(* IEC 61131-3 sources: ElnaAutomator/ExampleProject/build_USO_ecl (part 2) *)

  	END_CASE;
  END_IF;

  StrSw.Accident := inAccident.value AND inAccident.reliability;
  StrSw.Ns := inNs.value AND inNs.reliability;
  StrSw.Local := inLocal.value AND inLocal.reliability;
  StrSw.Distance := inDistance.value AND inDistance.reliability;
  StrSw.OpcCommandsDisabled := StrSw.inOpcCommandsDisabled;
  StrSw.offKNA := inoffKNA.value AND inoffKNA.reliability;

  (* ---- Формирование признака сдвига ---- *)

  getSdvig := FALSE;
  IF (StrSw.ISVALIDREF_cmdOn OR StrSw.ISVALIDREF_cmdOff) AND NOT StrSw.Local THEN
  	IF NOT (StrSw.CmdOn OR StrSw.CmdOff) THEN
                       IF (lastOnStatus <> StrSw.onStatus AND
  		(StrSw.onStatus <> _statusDualInput.STATUS_NOTDEFINED AND
                       StrSw.onStatus <> _statusDualInput.STATUS_ERROR)     AND
  		(lastOnStatus <> _statusDualInput.STATUS_NOTDEFINED   AND
                       lastOnStatus <> _statusDualInput.STATUS_ERROR))
                      THEN
  			getSdvig   := TRUE;
  		END_IF;
  	END_IF;
  END_IF;

  IF getSdvig THEN StrSw.sdvig:= TRUE; END_IF;

  sdvigReset(IN:=StrSw.sdvig, PT:=T#15S);

  IF sdvigReset.Q THEN StrSw.sdvig:=FALSE; END_IF;

  lastOnStatus := StrSw.onStatus;

  (* ---- Распаковка команды ---- *)
  _sunpackerCommand(command := StrSw.inCommand);
  	cmd := _sunpackerCommand.cmd;
  	source := _sunpackerCommand.source;

  (* ---- Обработка команды ---- *)
  IF cmd <> 0 AND lastCmd <> cmd and (((NOT StrSw.opcCommandsDisabled) AND source > 0) OR source = 0) then
  	CASE BYTE_TO_INT(cmd) OF
  	(*cmd_open*) 1 :
  			IF  StrSw.ISVALIDREF_cmdOn THEN StrSw.CmdOn := TRUE;
  				IF StrSw.ISVALIDREF_cmdOff THEN StrSw.CmdOff := FALSE; END_IF;
  			ELSIF  StrSw.ISVALIDREF_cmdOff THEN StrSw.CmdOff := FALSE;  END_IF;
  			errorCMDTimer(IN := false);
  			_commandErrorTimer := true;
  			StrSw.lastCmdIsOn := true;
  	(*cmd_close*) 2 :
  			IF StrSw.ISVALIDREF_cmdOff THEN StrSw.CmdOff := TRUE;
  				IF StrSw.ISVALIDREF_cmdOn THEN StrSw.CmdOn := FALSE; END_IF;
  			ELSIF StrSw.ISVALIDREF_cmdOn THEN StrSw.CmdOn := FALSE; END_IF;
  			errorCMDTimer(IN := false);
  			_commandErrorTimer := true;
  			StrSw.lastCmdIsOn := false;
  	(*cmd_reset*) 3 :    IF StrSw.ISVALIDREF_statOn OR StrSw.ISVALIDREF_statOff THEN
  			StrSw.CmdOn := FALSE;
  			StrSw.CmdOff := FALSE;
                                lastCmd := 0;
  			_commandErrorTimer := false;
  			StrSw.lastCmdIsOn := false;
                                 END_IF;
  	END_CASE;
  	source_for_Status := source;
  	cmd_for_Status := cmd;
  	command_error_for_Status := 0;
  END_IF;
  lastCmd := cmd;

  errorCMDTimer(In := _commandErrorTimer, PT :=T#10s);

  (* ---- алгоритм  для команды ВКЛючить ---- *)
  IF (StrSw.onStatus = _statusDualInput.STATUS_ON) and (StrSw.lastCmdIsOn) then
  	IF StrSw.ISVALIDREF_cmdOn AND StrSw.ISVALIDREF_cmdOff then  StrSw.cmdOn := false; END_IF;

  	 errorCMDTimer(In := false);
  	 _commandErrorTimer := false;
  	 cmd_for_Status := 0;
  	 source_for_Status := 0;
  END_IF;

  (* ---- off ---- *)
  IF (StrSw.onStatus = _statusDualInput.STATUS_OFF) and (NOT StrSw.lastCmdIsOn) then
  	IF StrSw.ISVALIDREF_cmdOn AND StrSw.ISVALIDREF_cmdOff then  StrSw.cmdOff := false; END_IF;

  	 errorCMDTimer(In := false);
  	 _commandErrorTimer := false;
  	 cmd_for_Status := 0;
  	 source_for_Status := 0;
  END_IF;

  (* ---- ошибка исполнения команды ---- *)
  if errorCMDTimer.Q and (cmd_for_Status <> 0) then
  	command_error_for_Status :=  cmd_for_Status;
  	_commandErrorTimer := false;
  	StrSw.CmdOn := false;
  	StrSw.CmdOff := false;
  	lastCmd := 0;
  end_if;

  (* ---- сброс ошибки команды ---- *)
  StrSw.CommandFault := command_error_for_Status <> 0;
  _errorReset(IN := command_error_for_Status <> 0, PT := T#5S);
  IF _errorReset.Q THEN
  	cmd_for_Status := 0;
  	source_for_Status := 0;
  	command_error_for_Status := 0;
  END_IF;

  outputsSets(in := (StrSw.ISVALIDREF_cmdOn and StrSw.cmdOn ) OR (StrSw.ISVALIDREF_cmdOff and StrSw.cmdOff), PT := T#2S);
  	IF NOT outputsSets.Q THEN
  		StrSw.BreakCmdOn := inBreakCmdOn._inversed AND inBreakCmdOn.reliability AND StrSw.ISVALIDREF_inBreakCmdOn;
  		StrSw.BreakCmdOff := inBreakCmdOff._inversed AND inBreakCmdOff.reliability AND StrSw.ISVALIDREF_inBreakCmdOff;
  	END_IF;

  cmdOn := StrSw.cmdOn;
  cmdOff:= StrSw.cmdOff;

  (* ---- формирование зашифрованного статуса для АРМа ---- *)
  StrSw.status := shl(BYTE_TO_DWORD(source_for_Status), 29)
  		OR shl(BYTE_TO_DWORD(cmd_for_Status), 26)
  		OR shl(BYTE_TO_DWORD(command_error_for_Status), 23)
  		OR shl(bool_to_DWORD(StrSw.sdvig), 22)
  		OR shl(bool_to_DWORD(StrSw.OpcCommandsDisabled), 21)
                      OR shl(BOOL_TO_DWORD(StrSw.offKNA), 17)
                      OR shl(bool_to_DWORD(StrSw.lastCmdIsOn), 14)
                      OR shl(BOOL_TO_DWORD(StrSw.BreakCmdOff), 13)
  		OR shl(BOOL_TO_DWORD(StrSw.BreakCmdOn), 12)
                      OR shl(BYTE_TO_DWORD(StrSw.basketStatus), 8)
  		OR shl(BOOL_TO_DWORD(StrSw.Distance), 6)
  		OR shl(BOOL_TO_DWORD(StrSw.Local), 5)
  		OR shl(BOOL_TO_DWORD(StrSw.Ns), 4)
                  	OR shl(BOOL_TO_DWORD(StrSw.Accident ),3)
  		OR BYTE_TO_DWORD(StrSw.onStatus);
END_FUNCTION_BLOCK

FUNCTION_BLOCK fb_singleOutput
  VAR_IN_OUT
    signal : BOOL;
    str_SO : struct_singleOutput;
  END_VAR
  VAR
    pulseTimer : TON;
    resetCmdTimer : TON;
    TON_Command : TON;
    source : BYTE;
    cmd : BYTE;
    lastCmd : BYTE;
    source_for_Status : BYTE;
    cmd_for_Status : BYTE;
    command_error_for_Status : BYTE;
    pulseTimerPriznak : BOOL;
    resetCmdTimerPriznak : BOOL;
    _sunpackerCommand : fb_sunpackerCommand;
  END_VAR

  str_SO.OpcCommandsDisabled := str_SO.inOpcCommandsDisabled;

  (* ---- Если управление с ВУ заблокировано, то передаем команду из алгоритма ---- *)
  IF str_SO.inOpcCommandsDisabled THEN
  	str_SO.inCommand := str_SO.inCommand_Alg;
  ELSE (* иначе передаем команду с АРМа*)
  	str_SO.inCommand := str_SO.inCommand_ARM;
  END_IF;

  (*Распаковка команды*)
  _sunpackerCommand(command := str_SO.inCommand);
  	cmd := _sunpackerCommand.cmd;
  	source := _sunpackerCommand.source;

  (*Обработка команды*)
  IF cmd <> 0 AND lastCmd <> cmd and (((NOT str_SO.OpcCommandsDisabled) AND source > 0) OR source = 0) then
  	CASE BYTE_TO_INT(cmd) OF
  	(*cmd_on*) 1 :
  			str_SO.Q := TRUE;
  			pulseTimer(IN := FALSE);
  			pulseTimerPriznak := FALSE;
  			resetCmdTimer(IN := FALSE);
  			resetCmdTimerPriznak := TRUE;
  	(*cmd_off*) 2 :
  			str_SO.Q := FALSE;
  			pulseTimer(IN := FALSE);
  			pulseTimerPriznak := FALSE;
  			resetCmdTimer(IN := FALSE);
  			resetCmdTimerPriznak := TRUE;
  	(*cmd_pulse*) 3 :
  			str_SO.Q := TRUE;
                                pulseTimer(IN := FALSE);
                                pulseTimerPriznak := TRUE;
  			resetCmdTimer(IN := FALSE);
                                resetCmdTimerPriznak := FALSE;
  	END_CASE;
  	source_for_Status := source;
  	cmd_for_Status := cmd;
  	command_error_for_Status := 0;
  END_IF;
  lastCmd := cmd;

  pulseTimer(IN := pulseTimerPriznak, PT := str_SO.wait_time);
  pulseTimer();
  IF pulseTimer.Q THEN
  	pulseTimer(IN := FALSE);
  	pulseTimerPriznak := FALSE;

  	str_SO.Q := FALSE;

  	source_for_Status := 0;
  	cmd_for_Status := 0;
  	command_error_for_Status := 0;
  END_IF;

  resetCmdTimer(IN := resetCmdTimerPriznak, PT := T#10S);
  resetCmdTimer();
  IF resetCmdTimer.Q THEN
  	resetCmdTimer(IN := FALSE);
  	resetCmdTimerPriznak := FALSE;

  	source_for_Status := 0;
  	cmd_for_Status := 0;
  	command_error_for_Status := 0;
  END_IF;

  signal:= str_SO.Q;

  (*TON_Command(IN:= (inCommand <> 0) AND (source = 0), PT:= T#2S);*)
      (*IF TON_Command.Q THEN*)
          (*inCommand := 0;*)
      (*END_IF;*)
  str_SO.status :=                           shl(BYTE_TO_DWORD(source_for_Status), 29)
  				OR shl(BYTE_TO_DWORD(cmd_for_Status), 26)
  				OR shl(BYTE_TO_DWORD(command_error_for_Status), 23)
  				OR shl(BOOL_TO_DWORD(str_SO.OpcCommandsDisabled), 21)
  				OR BOOL_TO_DWORD(str_SO.Q);
END_FUNCTION_BLOCK

FUNCTION_BLOCK fb_singleSignal
  VAR_INPUT
    signal : TYPE_ReliableBit;
  END_VAR
  VAR_IN_OUT
    str_SS : struct_singleSignal;
  END_VAR
  VAR
    TimerOn : TON;
    TimerOff : TOF;
  END_VAR

  str_SS.reliability:=signal.reliability;

  IF NOT str_SS.inverse THEN
  TimerOn(IN:=(signal.value AND str_SS.reliability AND NOT str_SS.Disabled_Sig), PT:=str_SS.DelayOn);
  ELSE
  TimerOn(IN:=(signal._inversed AND str_SS.reliability AND NOT str_SS.Disabled_Sig), PT:=str_SS.DelayOn);
  END_IF;

  TimerOff(IN:=TimerOn.Q, PT:=str_SS.DelayOff);

  str_SS.Q:=TimerOff.Q;

  str_SS.status:= SHL(BOOL_TO_DWORD(NOT str_SS.reliability), 15)
  	OR BOOL_TO_DWORD(str_SS.Q);
END_FUNCTION_BLOCK

FUNCTION_BLOCK Proc_Im
  VAR
    fb_Kran1 : fb_Kran;
    fb_Kran4 : fb_Kran;
    fb_Kran2 : fb_Kran;
    fb_Kran3 : fb_Kran;
    fb_Nu : fb_OilPump;
    fb_Nu2 : fb_OilPump;
    fb_Mv : fb_SectionSwitch;
    fb_SectionSwitch1 : fb_SectionSwitch;
    fb_Avom1 : fb_Switch;
    fb_Avom2 : fb_Switch;
    fb_Avom3 : fb_Switch;
    fb_Avom4 : fb_Switch;
    fb_So0 : fb_singleOutput;
    fb_So1 : fb_singleOutput;
    fb_So2 : fb_singleOutput;
    fb_So3 : fb_singleOutput;
    fb_So4 : fb_singleOutput;
    fb_So5 : fb_singleOutput;
    fb_So6 : fb_singleOutput;
    fb_So7 : fb_singleOutput;
    fb_SI0 : fb_singleSignal;
    fb_SI1 : fb_singleSignal;
    fb_SI2 : fb_singleSignal;
    fb_SI3 : fb_singleSignal;
    fb_SI4 : fb_singleSignal;
    fb_SI5 : fb_singleSignal;
    fb_SI6 : fb_singleSignal;
  END_VAR
  VAR_EXTERNAL
    di : DiConfig;
    od : DoConfig;
    Im : ImConfig;
  END_VAR

  fb_Kran1(statOn := di.Di.bits[1]._inversed,
  statOn_reliability := di.Di.bits[1].reliability,
  statOff := di.Di.bits[2]._inversed,
  statOff_reliability := di.Di.bits[2].reliability,
  cmdOn := od.Do1.bits[1],
  cmdOff := od.Do2.bits[0],
  inDp := di.Di1.bits[1],
  inSo := di.Di.bits[3],
  inSz := di.Di.bits[2],
  strKr := Im.Kran1);

  fb_Kran4(statOn := di.Di1.bits[2]._inversed,
  statOn_reliability := di.Di1.bits[2].reliability,
  statOff := di.Di2.bits[2]._inversed,
  statOff_reliability := di.Di2.bits[2].reliability,
  cmdOn := od.Do3.bits[2],
  cmdOff := od.Do1.bits[2],
  inDp := di.Di.bits[2],
  inSo := di.Di2.bits[3],
  inSz := di.Di1.bits[1],
  strKr := Im.Kran4);

  fb_Kran2(statOn := di.Di2.bits[3].value,
  statOn_reliability := di.Di2.bits[3].reliability,
  statOff := di.Di3.bits[1].value,
  statOff_reliability := di.Di3.bits[1].reliability,
  cmdOn := od.Do3.bits[3],
  cmdOff := od.Do2.bits[3],
  inDp := di.Di4.bits[3],
  inSo := di.Di1.bits[1],
  inSz := di.Di1.bits[2],
  strKr := Im.Kran2);

  fb_Kran3(statOn := di.Di3.bits[4]._inversed,
  statOn_reliability := di.Di3.bits[4].reliability,
  statOff := di.Di4.bits[3]._inversed,
  statOff_reliability := di.Di4.bits[3].reliability,
  cmdOn := od.Do2.bits[4],
  cmdOff := od.Do3.bits[4],
  inDp := di.Di4.bits[4],
  inSo := di.Di1.bits[2],
  inSz := di.Di4.bits[3],
  strKr := Im.Kran3);

  fb_Nu(statOn := di.Di.bits[1]._inversed,
  statOn_reliability := di.Di.bits[1].reliability,
  statOff := di.Di.bits[2]._inversed,
  statOff_reliability := di.Di.bits[2].reliability,
  cmdOn := od.Do2.bits[1],
  cmdOff := od.Do1.bits[0],
  inBreakCmdOn := di.Di.bits[3],
  inBreakCmdOff := di.Di1.bits[4],
  StrSw := Im.Nu);

  fb_Nu2(statOn := di.Di2.bits[2].value,
  statOn_reliability := di.Di2.bits[2].reliability,
  statOff := di.Di3.bits[3].value,
  statOff_reliability := di.Di3.bits[3].reliability,
  cmdOn := od.Do4.bits[3],
  cmdOff := od.Do1.bits[4],
  inBreakCmdOn := di.Di.bits[4],
  inBreakCmdOff := di.Di1.bits[3],
  StrSw := Im.Nu2);

  fb_Avom1(statOn := di.Di.bits[1].value,
  statOn_reliability := di.Di.bits[1].reliability,
  statOff := di.Di1.bits[2].value,
  statOff_reliability := di.Di1.bits[2].reliability,
  cmdOn := od.Do1.bits[1],
  cmdOff := od.Do1.bits[0],
  inBreakCmdOn := di.Di1.bits[2],
  inBreakCmdOff := di.Di.bits[2],
  StrSw := Im.Avom1);

  fb_Avom2(statOn := di.Di3.bits[2]._inversed,
  statOn_reliability := di.Di3.bits[2].reliability,
  statOff := di.Di.bits[2]._inversed,
  statOff_reliability := di.Di.bits[2].reliability,
  cmdOn := od.Do4.bits[3],
  cmdOff := od.Do2.bits[1],
  inBreakCmdOn := di.Di1.bits[3],
  inBreakCmdOff := di.Di1.bits[3],
  StrSw := Im.Avom2);

  fb_Avom3(statOn := di.Di1.bits[3]._inversed,
  statOn_reliability := di.Di1.bits[3].reliability,
  statOff := di.Di2.bits[3]._inversed,
  statOff_reliability := di.Di2.bits[3].reliability,
  cmdOn := od.Do1.bits[5],
  cmdOff := od.Do3.bits[3],
  inBreakCmdOn := di.Di3.bits[4],
  inBreakCmdOff := di.Di2.bits[4],
  StrSw := Im.Avom3);

  fb_Avom4(statOn := di.Di.bits[4]._inversed,
  statOn_reliability := di.Di.bits[4].reliability,
  statOff := di.Di.bits[4]._inversed,
  statOff_reliability := di.Di.bits[4].reliability,
  cmdOn := od.Do2.bits[4],
  cmdOff := od.Do3.bits[4],
  inBreakCmdOn := di.Di3.bits[5],
  inBreakCmdOff := di.Di4.bits[5],
  StrSw := Im.Avom4);

  fb_Mv(statOn := di.Di.bits[1]._inversed,
  statOn_reliability := di.Di.bits[1].reliability,
  statOff := di.Di.bits[2]._inversed,
  statOff_reliability := di.Di.bits[2].reliability,
  cmdOn := od.Do2.bits[1],
  cmdOff := od.Do2.bits[0],
  inBreakCmdOn := di.Di3.bits[4],
  inBreakCmdOff := di.Di4.bits[3],
  basketRolledin := di.Di.bits[2],
  basketRolledout := di.Di.bits[3],
  basketTest := di.Di1.bits[3],
  StrSw := Im.Mv);

  fb_SectionSwitch1(StrSw := Im.SectionSwitch1);

  fb_SI0(signal := di.Di1.bits[1], str_SS := Im.SingleSignals.SI0);

  fb_SI1(signal := di.Di1.bits[2], str_SS := Im.SingleSignals.SI1);

  fb_SI2(signal := di.Di.bits[3], str_SS := Im.SingleSignals.SI2);

  fb_SI3(signal := di.Di1.bits[4], str_SS := Im.SingleSignals.SI3);

  fb_SI4(signal := di.Di3.bits[5], str_SS := Im.SingleSignals.SI4);

  fb_SI5(signal := di.Di3.bits[6], str_SS := Im.SingleSignals.SI5);

  fb_SI6(signal := di.Di4.bits[7], str_SS := Im.SingleSignals.SI6);

  fb_So0(signal := od.Do1.bits[1], str_SO := Im.SingleOutputs.So0);

  fb_So1(signal := od.Do2.bits[2], str_SO := Im.SingleOutputs.So1);

  fb_So2(signal := od.Do3.bits[3], str_SO := Im.SingleOutputs.So2);

  fb_So3(signal := od.Do1.bits[4], str_SO := Im.SingleOutputs.So3);

  fb_So4(signal := od.Do2.bits[5], str_SO := Im.SingleOutputs.So4);

  fb_So5(signal := od.Do1.bits[6], str_SO := Im.SingleOutputs.So5);

  fb_So6(signal := od.Do1.bits[7], str_SO := Im.SingleOutputs.So6);

  fb_So7(signal := od.Do2.bits[8], str_SO := Im.SingleOutputs.So7);
END_FUNCTION_BLOCK

FUNCTION_BLOCK Proc_Do_Init
  VAR_INPUT
    init : BOOL;
  END_VAR
  VAR
    stDO_Ini : fb_DO_Init;
    inits : UINT;
  END_VAR
  VAR_INPUT
    initiales : UINT;
  END_VAR
  VAR_EXTERNAL
    od : DoConfig;
  END_VAR

  inits := 0;

  stDO_Ini(data_Ini := TRUE, imit := FALSE, strDO := od.Do1);
  inits := inits + BOOL_TO_UINT(stDO_Ini.Init);

  stDO_Ini(data_Ini := TRUE, imit := FALSE, strDO := od.Do2);
  inits := inits + BOOL_TO_UINT(stDO_Ini.Init);

  stDO_Ini(data_Ini := TRUE, imit := FALSE, strDO := od.Do3);
  inits := inits + BOOL_TO_UINT(stDO_Ini.Init);

  stDO_Ini(data_Ini := TRUE, imit := FALSE, strDO := od.Do4);
  inits := inits + BOOL_TO_UINT(stDO_Ini.Init);

  stDO_Ini(data_Ini := TRUE, imit := FALSE, strDO := od.Do5);
  inits := inits + BOOL_TO_UINT(stDO_Ini.Init);

  initiales := 0;
  IF init THEN initiales := inits; END_IF;
END_FUNCTION_BLOCK

FUNCTION_BLOCK Opc_Im_set
  VAR_EXTERNAL
    Im : ImConfig;
    Im_Kran1_status : UDINT;
    Im_Kran4_status : UDINT;
    Im_Kran2_status : UDINT;
    Im_Kran3_status : UDINT;
    Im_Nu_status : UDINT;
    Im_Nu2_status : UDINT;
    Im_Avom1_status : UDINT;
    Im_Avom2_status : UDINT;
    Im_Avom3_status : UDINT;
    Im_Avom4_status : UDINT;
    Im_Mv_status : UDINT;
    Im_SectionSwitch1_status : UDINT;
    Im_SingleSignals_SI0_status : UDINT;
    Im_SingleSignals_SI1_status : UDINT;
    Im_SingleSignals_SI2_status : UDINT;
    Im_SingleSignals_SI3_status : UDINT;
    Im_SingleSignals_SI4_status : UDINT;
    Im_SingleSignals_SI5_status : UDINT;
    Im_SingleSignals_SI6_status : UDINT;
  END_VAR

  Im_Kran1_status := DWORD_TO_UDINT(Im.Kran1.status);

  Im_Kran4_status := DWORD_TO_UDINT(Im.Kran4.status);

  Im_Kran2_status := DWORD_TO_UDINT(Im.Kran2.status);

  Im_Kran3_status := DWORD_TO_UDINT(Im.Kran3.status);

  Im_Nu_status := DWORD_TO_UDINT(Im.Nu.status);

  Im_Nu2_status := DWORD_TO_UDINT(Im.Nu2.status);

  Im_Avom1_status := DWORD_TO_UDINT(Im.Avom1.status);

  Im_Avom2_status := DWORD_TO_UDINT(Im.Avom2.status);

  Im_Avom3_status := DWORD_TO_UDINT(Im.Avom3.status);

  Im_Avom4_status := DWORD_TO_UDINT(Im.Avom4.status);

  Im_Mv_status := DWORD_TO_UDINT(Im.Mv.status);

  Im_SectionSwitch1_status := DWORD_TO_UDINT(Im.SectionSwitch1.status);

  Im_SingleSignals_SI0_status := DWORD_TO_UDINT(Im.SingleSignals.SI0.status);

  Im_SingleSignals_SI1_status := DWORD_TO_UDINT(Im.SingleSignals.SI1.status);

  Im_SingleSignals_SI2_status := DWORD_TO_UDINT(Im.SingleSignals.SI2.status);

  Im_SingleSignals_SI3_status := DWORD_TO_UDINT(Im.SingleSignals.SI3.status);

  Im_SingleSignals_SI4_status := DWORD_TO_UDINT(Im.SingleSignals.SI4.status);

  Im_SingleSignals_SI5_status := DWORD_TO_UDINT(Im.SingleSignals.SI5.status);

  Im_SingleSignals_SI6_status := DWORD_TO_UDINT(Im.SingleSignals.SI6.status);
END_FUNCTION_BLOCK

FUNCTION_BLOCK Opc_Im_get
  VAR_EXTERNAL
    Im : ImConfig;
    Im_Kran1_inCommand_ARM : UINT;
    Im_Kran4_inCommand_ARM : UINT;
    Im_Kran2_inCommand_ARM : UINT;
    Im_Kran3_inCommand_ARM : UINT;
    Im_Nu_inCommand_ARM : UINT;
    Im_Nu2_inCommand_ARM : UINT;
    Im_Avom1_inCommand_ARM : UINT;
    Im_Avom2_inCommand_ARM : UINT;
    Im_Avom3_inCommand_ARM : UINT;
    Im_Avom4_inCommand_ARM : UINT;
    Im_Mv_inCommand_ARM : UINT;
    Im_SectionSwitch1_inCommand_ARM : UINT;
  END_VAR

  Im.Kran1.inCommand_ARM := UINT_TO_WORD(Im_Kran1_inCommand_ARM);

  Im.Kran4.inCommand_ARM := UINT_TO_WORD(Im_Kran4_inCommand_ARM);

  Im.Kran2.inCommand_ARM := UINT_TO_WORD(Im_Kran2_inCommand_ARM);

  Im.Kran3.inCommand_ARM := UINT_TO_WORD(Im_Kran3_inCommand_ARM);

  Im.Nu.inCommand_ARM := UINT_TO_WORD(Im_Nu_inCommand_ARM);

  Im.Nu2.inCommand_ARM := UINT_TO_WORD(Im_Nu2_inCommand_ARM);

  Im.Avom1.inCommand_ARM := UINT_TO_WORD(Im_Avom1_inCommand_ARM);

  Im.Avom2.inCommand_ARM := UINT_TO_WORD(Im_Avom2_inCommand_ARM);

  Im.Avom3.inCommand_ARM := UINT_TO_WORD(Im_Avom3_inCommand_ARM);

  Im.Avom4.inCommand_ARM := UINT_TO_WORD(Im_Avom4_inCommand_ARM);

  Im.Mv.inCommand_ARM := UINT_TO_WORD(Im_Mv_inCommand_ARM);

  Im.SectionSwitch1.inCommand_ARM := UINT_TO_WORD(Im_SectionSwitch1_inCommand_ARM);
END_FUNCTION_BLOCK

FUNCTION_BLOCK Opc_Ai_set
  VAR_EXTERNAL
    Ai : AiConfig;
    AI_A1_HW : LREAL;
    AI_A1_HA : LREAL;
    AI_A1_LA : LREAL;
    AI_A1_LW : LREAL;
    AI_A1_HL : LREAL;
    AI_A1_LL : LREAL;
    AI_A1_value : LREAL;
    AI_A1_status : UDINT;
    AI_A2_HW : LREAL;
    AI_A2_HA : LREAL;
    AI_A2_LA : LREAL;
    AI_A2_LW : LREAL;
    AI_A2_HL : LREAL;
    AI_A2_LL : LREAL;
    AI_A2_value : LREAL;
    AI_A2_status : UDINT;
  END_VAR

  AI_A1_HW := Ai.A1.HW;
  AI_A1_HA := Ai.A1.HA;
  AI_A1_LA := Ai.A1.LA;
  AI_A1_LW := Ai.A1.LW;
  AI_A1_LL := Ai.A1.LL;
  AI_A1_HL := Ai.A1.HL;
  AI_A1_value := Ai.A1.value;
  AI_A1_status := DWORD_TO_UDINT(Ai.A1.status);

  AI_A2_HW := Ai.A2.HW;
  AI_A2_HA := Ai.A2.HA;
  AI_A2_LA := Ai.A2.LA;
  AI_A2_LW := Ai.A2.LW;
  AI_A2_LL := Ai.A2.LL;
  AI_A2_HL := Ai.A2.HL;
  AI_A2_value := Ai.A2.value;
  AI_A2_status := DWORD_TO_UDINT(Ai.A2.status);
END_FUNCTION_BLOCK

FUNCTION_BLOCK Proc_Do
  VAR
    fb_Do1 : fb_DOSourceMlp;
    fb_Do2 : fb_DOSourceMlp;
    fb_Do3 : fb_DOSourceMlp;
    fb_Do4 : fb_DOSourceMlp;
    fb_Do5 : fb_DOSourceMlp;
  END_VAR
  VAR_EXTERNAL
    od : DoConfig;
    arDOUT_0 : TWordData;
    arDOUT_1 : TWordData;
    arDOUT_2 : TWordData;
    arDOUT_3 : TWordData;
    arDOUT_4 : TWordData;
    DO_0_wValue : UINT;
    DO_1_wValue : UINT;
    DO_2_wValue : UINT;
    DO_3_wValue : UINT;
    DO_4_wValue : UINT;
    arERR_1 : TItemDIN;
    arERR_2 : TItemDIN;
    arERR_3 : TItemDIN;
    arERR_4 : TItemDIN;
    arERR_5 : TItemDIN;
  END_VAR

  fb_Do1(arDout := arDOUT_0, strDO := od.Do1, err_mod := arERR_1);
  DO_0_wValue := arDOUT_0.wValue;

  fb_Do2(arDout := arDOUT_1, strDO := od.Do2, err_mod := arERR_2);
  DO_1_wValue := arDOUT_1.wValue;

  fb_Do3(arDout := arDOUT_2, strDO := od.Do3, err_mod := arERR_3);
  DO_2_wValue := arDOUT_2.wValue;

  fb_Do4(arDout := arDOUT_3, strDO := od.Do4, err_mod := arERR_4);
  DO_3_wValue := arDOUT_3.wValue;

  fb_Do5(arDout := arDOUT_4, strDO := od.Do5, err_mod := arERR_5);
  DO_4_wValue := arDOUT_4.wValue;

  (*gpio_out not initialized*)
END_FUNCTION_BLOCK

FUNCTION_BLOCK Proc_Di_Init
  VAR_INPUT
    init : BOOL;
  END_VAR
  VAR
    stDI_Ini : fb_DI_Init;
    inits : UINT;
  END_VAR
  VAR_INPUT
    initiales : UINT;
  END_VAR
  VAR_EXTERNAL
    di : DiConfig;
  END_VAR

  inits := 0;

  stDI_Ini(data_Ini := TRUE, imit := FALSE, strDI := di.Di);
  inits := inits + BOOL_TO_UINT(stDI_Ini.Init);

  stDI_Ini(data_Ini := TRUE, imit := FALSE, strDI := di.Di1);
  inits := inits + BOOL_TO_UINT(stDI_Ini.Init);

  stDI_Ini(data_Ini := TRUE, imit := FALSE, strDI := di.Di2);
  inits := inits + BOOL_TO_UINT(stDI_Ini.Init);

  stDI_Ini(data_Ini := TRUE, imit := FALSE, strDI := di.Di3);
  inits := inits + BOOL_TO_UINT(stDI_Ini.Init);

  stDI_Ini(data_Ini := TRUE, imit := FALSE, strDI := di.Di4);
  inits := inits + BOOL_TO_UINT(stDI_Ini.Init);

  initiales := 0;
  IF init THEN initiales := inits; END_IF;
END_FUNCTION_BLOCK

FUNCTION_BLOCK Opc_Protections_set
  VAR_EXTERNAL
    Protections : ProtectionsConfig;
    Protections_Ap1_status : UDINT;
    Protections_AiP1_status : UDINT;
    Protections_AiP2_status : UDINT;
    Protections_AiP3_status : UDINT;
    Protections_DiP1_status : UDINT;
    Protections_DiP2_status : UDINT;
    Protections_DiP3_status : UDINT;
    Protections_DiP4_status : UDINT;
    Protections_DiP5_status : UDINT;
  END_VAR

  Protections_Ap1_status := DWORD_TO_UDINT(Protections.Ap1.status);

  Protections_AiP1_status := DWORD_TO_UDINT(Protections.AiP1.status);

  Protections_AiP2_status := DWORD_TO_UDINT(Protections.AiP2.status);

  Protections_AiP3_status := DWORD_TO_UDINT(Protections.AiP3.status);

  Protections_DiP1_status := DWORD_TO_UDINT(Protections.DiP1.status);

  Protections_DiP2_status := DWORD_TO_UDINT(Protections.DiP2.status);

  Protections_DiP3_status := DWORD_TO_UDINT(Protections.DiP3.status);

  Protections_DiP4_status := DWORD_TO_UDINT(Protections.DiP4.status);

  Protections_DiP5_status := DWORD_TO_UDINT(Protections.DiP5.status);
END_FUNCTION_BLOCK

FUNCTION_BLOCK Opc_Protections_get
  VAR_EXTERNAL
    Protections : ProtectionsConfig;
    Protections_Ap1_inCommand_ARM : UINT;
    Protections_AiP1_inCommand_ARM : UINT;
    Protections_AiP2_inCommand_ARM : UINT;
    Protections_AiP3_inCommand_ARM : UINT;
    Protections_DiP1_inCommand_ARM : UINT;
    Protections_DiP2_inCommand_ARM : UINT;
    Protections_DiP3_inCommand_ARM : UINT;
    Protections_DiP4_inCommand_ARM : UINT;
    Protections_DiP5_inCommand_ARM : UINT;
  END_VAR

  Protections.Ap1.inCommand_ARM := UINT_TO_WORD(Protections_Ap1_inCommand_ARM);

  Protections.AiP1.inCommand_ARM := UINT_TO_WORD(Protections_AiP1_inCommand_ARM);

  Protections.AiP2.inCommand_ARM := UINT_TO_WORD(Protections_AiP2_inCommand_ARM);

  Protections.AiP3.inCommand_ARM := UINT_TO_WORD(Protections_AiP3_inCommand_ARM);

  Protections.DiP1.inCommand_ARM := UINT_TO_WORD(Protections_DiP1_inCommand_ARM);

  Protections.DiP2.inCommand_ARM := UINT_TO_WORD(Protections_DiP2_inCommand_ARM);

  Protections.DiP3.inCommand_ARM := UINT_TO_WORD(Protections_DiP3_inCommand_ARM);

  Protections.DiP4.inCommand_ARM := UINT_TO_WORD(Protections_DiP4_inCommand_ARM);

  Protections.DiP5.inCommand_ARM := UINT_TO_WORD(Protections_DiP5_inCommand_ARM);
END_FUNCTION_BLOCK

FUNCTION_BLOCK fb_DiSourceMlp
  VAR_INPUT
    arDIN : TItemDIN;
    err_mod : TItemDIN;
  END_VAR
  VAR_IN_OUT
    strDI : struct_DI;
  END_VAR
  VAR_OUTPUT
    Bounce : BOOL;
  END_VAR
  VAR
    _value : WORD;
    _reliability : BOOL;
    bitNumber : INT;
    bitNum : INT;
  END_VAR

  strDI.blConnect := (*((UINT_TO_WORD(arDIN.wFlags) = 1472) and*) (UINT_TO_WORD(err_mod.wValue) = 20) and (UINT_TO_WORD(err_mod.wFlags) = 192);
  Bounce := (UINT_TO_WORD(arDIN.wFlags) AND 16#0020) <> 0;

  If NOT strDI.imit THEN
  _value:=UINT_TO_WORD(arDIN.wValue);

      IF strDI.blConnect THEN
            strDI.reliability:=0;
            strDI.value:=0;
  	FOR bitNumber:=0 TO 7 BY 1 DO

  		_reliability:=WORD_TO_BOOL(SHR(_value, bitNumber*2) AND 16#2);
  		strDI.reliability:=strDI.reliability OR SHL(BOOL_TO_WORD(_reliability),bitNumber);
  		IF _reliability THEN
  			strDI.value:=strDI.value OR SHL((SHR(_value, bitNumber*2) AND 16#1),bitNumber);
  		END_IF;
  	END_FOR;
      ELSE
  	strDI.reliability := 0;
      END_IF;

      FOR bitNum:=0 TO 15 BY 1 DO
  	          strDI.bits[bitNum].reliability :=WORD_TO_BOOL(SHR(strDI.reliability, bitNum) AND 16#1);
  	IF strDI.bits[bitNum].reliability THEN
  		strDI.bits[bitNum].value :=WORD_TO_BOOL(SHR(strDI.value, bitNum) AND 16#1);
                      strDI.bits[bitNum]._inversed :=NOT strDI.bits[bitNum].value;
  	END_IF;
      END_FOR;

  END_IF;
END_FUNCTION_BLOCK

FUNCTION_BLOCK Proc_Protections_Init
  VAR_INPUT
    init : BOOL;
  END_VAR
  VAR
    stDIp_Ini : fb_DiProtection_Init;
    stAIp_Ini : fb_AiProtection_Init;
    inits : UINT;
  END_VAR
  VAR_INPUT
    initiales : UINT;
  END_VAR
  VAR_EXTERNAL
    Protections : ProtectionsConfig;
  END_VAR
  VAR
    _ProtectionTags : TYPE_ProtectionTags;
    _StatusAi : TYPE_StatusAi;
  END_VAR

  inits := 0;

  stAIp_Ini(data_Ini := TRUE, delay := T#1S, inTag := _ProtectionTags.AOS, inRunOnStart := TRUE,
  controlLimit := _StatusAi.LA, str_AIp := Protections.Ap1);
  inits := inits + BOOL_TO_UINT(stAIp_Ini.Init);

  stAIp_Ini(data_Ini := TRUE, delay := T#2S, inTag := _ProtectionTags.AOS, inRunOnStart := FALSE,
  controlLimit := _StatusAi.HA, str_AIp := Protections.AiP1);
  inits := inits + BOOL_TO_UINT(stAIp_Ini.Init);

  stAIp_Ini(data_Ini := TRUE, delay := T#3S, inTag := _ProtectionTags.AOS, inRunOnStart := TRUE,
  controlLimit := _StatusAi.LA, str_AIp := Protections.AiP2);
  inits := inits + BOOL_TO_UINT(stAIp_Ini.Init);

  stAIp_Ini(data_Ini := TRUE, delay := T#4S, inTag := _ProtectionTags.AOS, inRunOnStart := FALSE,
  controlLimit := _StatusAi.HA, str_AIp := Protections.AiP3);
  inits := inits + BOOL_TO_UINT(stAIp_Ini.Init);

  stDIp_Ini(data_Ini := TRUE, delay := T#1S, inTag := _ProtectionTags.AOS, inRunOnStart := TRUE, str_DIp := Protections.DiP1);
  inits := inits + BOOL_TO_UINT(stDIp_Ini.Init);

  stDIp_Ini(data_Ini := TRUE, delay := T#2S, inTag := _ProtectionTags.AOS, inRunOnStart := TRUE, str_DIp := Protections.DiP2);
  inits := inits + BOOL_TO_UINT(stDIp_Ini.Init);

  stDIp_Ini(data_Ini := TRUE, delay := T#3S, inTag := _ProtectionTags.AOS, inRunOnStart := TRUE, str_DIp := Protections.DiP3);
  inits := inits + BOOL_TO_UINT(stDIp_Ini.Init);

  stDIp_Ini(data_Ini := TRUE, delay := T#4S, inTag := _ProtectionTags.AOS, inRunOnStart := FALSE, str_DIp := Protections.DiP4);
  inits := inits + BOOL_TO_UINT(stDIp_Ini.Init);

  stDIp_Ini(data_Ini := TRUE, delay := T#5S, inTag := _ProtectionTags.AOS, inRunOnStart := FALSE, str_DIp := Protections.DiP5);
  inits := inits + BOOL_TO_UINT(stDIp_Ini.Init);

  IF init THEN initiales := inits; END_IF;
END_FUNCTION_BLOCK

FUNCTION_BLOCK Proc_Di
  VAR
    fb_Di : fb_DiSourceMlp;
    fb_Di1 : fb_DiSourceMlp;
    fb_Di2 : fb_DiSourceMlp;
    fb_Di3 : fb_DiSourceMlp;
    fb_Di4 : fb_DiSourceMlp;
  END_VAR
  VAR_EXTERNAL
    di : DiConfig;
    arDIN_0 : TItemDIN;
    arDIN_1 : TItemDIN;
    arDIN_2 : TItemDIN;
    arDIN_3 : TItemDIN;
    arDIN_4 : TItemDIN;
    DI_0_1_wValue : UDINT;
    DI_2_3_wValue : UDINT;
    arERR_1 : TItemDIN;
    arERR_2 : TItemDIN;
    arERR_3 : TItemDIN;
    arERR_4 : TItemDIN;
    arERR_5 : TItemDIN;
  END_VAR

  fb_Di(arDIN := arDIN_0, strDI := di.Di, err_mod := arERR_1);
  fb_Di1(arDIN := arDIN_1, strDI := di.Di1, err_mod := arERR_2);
  DI_0_1_wValue := DIwValue_Diag(arDIN_0.wValue, arDIN_1.wValue);

  fb_Di2(arDIN := arDIN_2, strDI := di.Di2, err_mod := arERR_3);
  fb_Di3(arDIN := arDIN_3, strDI := di.Di3, err_mod := arERR_4);
  DI_2_3_wValue := DIwValue_Diag(arDIN_2.wValue, arDIN_3.wValue);

  fb_Di4(arDIN := arDIN_4, strDI := di.Di4, err_mod := arERR_5);
END_FUNCTION_BLOCK

PROGRAM program0
  VAR
    Var0 : DINT;
  END_VAR

  Var0 := 1;
END_PROGRAM

CONFIGURATION config1
  VAR_GLOBAL
    systime_s AT %IL0.10.10 : ULINT;
    systime_ns AT %IL0.10.11 : ULINT;
    current_retrieve_us AT %IL0.10.12 : ULINT;
    current_config_us AT %IL0.10.13 : ULINT;
    current_publish_us AT %IL0.10.14 : ULINT;
    current_run_us AT %IL0.10.15 : ULINT;
    max_retrieve_us AT %QL0.10.16 : ULINT;
    max_config_us AT %QL0.10.17 : ULINT;
    max_publish_us AT %QL0.10.18 : ULINT;
    plc_run_number AT %IL0.10.19 : ULINT;
    arAIN_0 : TItemAIN;
    arAIN_1 : TItemAIN;
    arAIN_2 : TItemAIN;
    arAIN_3 : TItemAIN;
    arAIN_4 : TItemAIN;
    arAIN_5 : TItemAIN;
    arAIN_6 : TItemAIN;
    arAIN_7 : TItemAIN;
    arAIN_8 : TItemAIN;
    arAIN_9 : TItemAIN;
    arAIN_10 : TItemAIN;
    arAIN_11 : TItemAIN;
    arAIN_12 : TItemAIN;
    arAIN_13 : TItemAIN;
    arAIN_14 : TItemAIN;
    arAIN_15 : TItemAIN;
    arAIN_16 : TItemAIN;
    arAIN_17 : TItemAIN;
    arAIN_18 : TItemAIN;
    arAIN_19 : TItemAIN;
    arAIN_20 : TItemAIN;
    arAIN_21 : TItemAIN;
    arAIN_22 : TItemAIN;
    arAIN_23 : TItemAIN;
    arAIN_24 : TItemAIN;
    arAIN_25 : TItemAIN;
    arAIN_26 : TItemAIN;
    arAIN_27 : TItemAIN;
    arAIN_28 : TItemAIN;
    arAIN_29 : TItemAIN;
    arAIN_30 : TItemAIN;
    arAIN_31 : TItemAIN;
    arAIN_32 : TItemAIN;
    arAIN_33 : TItemAIN;
    arAIN_34 : TItemAIN;
    arAIN_35 : TItemAIN;
    arAIN_36 : TItemAIN;
    arAIN_37 : TItemAIN;
    arAIN_38 : TItemAIN;
    arAIN_39 : TItemAIN;
    arAIN_40 : TItemAIN;
    arAIN_41 : TItemAIN;
    arAIN_42 : TItemAIN;
    arAIN_43 : TItemAIN;
    arAIN_44 : TItemAIN;
    arAIN_45 : TItemAIN;
    arAIN_46 : TItemAIN;
    arAIN_47 : TItemAIN;
    arAIN_48 : TItemAIN;
    arAIN_49 : TItemAIN;
    arAIN_50 : TItemAIN;
    arAIN_51 : TItemAIN;
    arAIN_52 : TItemAIN;
    arAIN_53 : TItemAIN;
    arAIN_54 : TItemAIN;
    arAIN_55 : TItemAIN;
    arAIN_56 : TItemAIN;
    arAIN_57 : TItemAIN;
    arAIN_58 : TItemAIN;
    arAIN_59 : TItemAIN;
    arAIN_60 : TItemAIN;
    arAIN_61 : TItemAIN;
    arAIN_62 : TItemAIN;
    arAIN_63 : TItemAIN;
    arAIN_64 : TItemAIN;
    arAIN_65 : TItemAIN;
    arAIN_66 : TItemAIN;
    arAIN_67 : TItemAIN;
    arAIN_68 : TItemAIN;
    arAIN_69 : TItemAIN;
    arAIN_70 : TItemAIN;
    arAIN_71 : TItemAIN;
    arAIN_72 : TItemAIN;
    arAIN_73 : TItemAIN;
    arAIN_74 : TItemAIN;
    arAIN_75 : TItemAIN;
    arAIN_76 : TItemAIN;
    arAIN_77 : TItemAIN;
    arAIN_78 : TItemAIN;
    arAIN_79 : TItemAIN;
    arDIN_0 : TItemDIN;
    arDIN_1 : TItemDIN;
    arDIN_2 : TItemDIN;
    arDIN_3 : TItemDIN;
    arDIN_4 : TItemDIN;
    arDIN_5 : TItemDIN;
    arDIN_6 : TItemDIN;
    arDIN_7 : TItemDIN;
    arDIN_8 : TItemDIN;
    arDIN_9 : TItemDIN;
    arDIN_10 : TItemDIN;
    arDIN_11 : TItemDIN;
    arDIN_12 : TItemDIN;
    arDIN_13 : TItemDIN;
    arDIN_14 : TItemDIN;
    arDIN_15 : TItemDIN;
    arDIN_16 : TItemDIN;
    arDIN_17 : TItemDIN;
    arDIN_18 : TItemDIN;
    arDIN_19 : TItemDIN;
    arDIN_20 : TItemDIN;
    arDIN_21 : TItemDIN;
    arAOUT_0 : TDoubleData;
    arAOUT_1 : TDoubleData;
    arDOUT_0 : TWordData;
    arDOUT_1 : TWordData;
    arDOUT_2 : TWordData;
    arDOUT_3 : TWordData;
    arDOUT_4 : TWordData;
    arDOUT_5 : TWordData;
    arDOUT_6 : TWordData;
    arDOUT_7 : TWordData;
    arDOUT_8 : TWordData;
    arDOUT_9 : TWordData;
    arDOUT_10 : TWordData;
    arDOUT_11 : TWordData;
    arDOUT_12 : TWordData;
    arDOUT_13 : TWordData;
    arDOUT_66 : TWordData;
    arERR_0 : TItemDIN;
    arERR_1 : TItemDIN;
    arERR_2 : TItemDIN;
    arERR_3 : TItemDIN;
    arERR_4 : TItemDIN;
    arERR_5 : TItemDIN;
    arERR_6 : TItemDIN;
    arERR_7 : TItemDIN;
    arERR_8 : TItemDIN;
    arERR_9 : TItemDIN;
    arERR_10 : TItemDIN;
    arERR_11 : TItemDIN;
    arERR_12 : TItemDIN;
    arERR_13 : TItemDIN;
    arERR_14 : TItemDIN;
    arERR_15 : TItemDIN;
    arERR_16 : TItemDIN;
    arERR_17 : TItemDIN;
    arERR_18 : TItemDIN;
    arERR_19 : TItemDIN;
    arERR_20 : TItemDIN;
    arERR_21 : TItemDIN;
    arERR_22 : TItemDIN;
    arERR_23 : TItemDIN;
    arERR_24 : TItemDIN;
    arERR_25 : TItemDIN;
    arERR_66 : TItemDIN;
    arRelSt_0 : TItemDIN;
  END_VAR

  RESOURCE resource1 ON PLC
    VAR_GLOBAL CONSTANT
      gMaint_Time : REAL;
    END_VAR
    VAR_GLOBAL
      Ai : AiConfig;
      Im : ImConfig;
      di : DiConfig;
      od : DoConfig;
      cur_Cycle : REAL;
      gStart_Tmr : REAL;
    END_VAR
    VAR_GLOBAL CONSTANT
      req_Cycle : REAL := 0.02;
    END_VAR
    VAR_GLOBAL
      gF_T_100mSec : BOOL;
      gT_1Sec : BOOL;
      gF_T_1Sec : BOOL;
      gT_1Min : BOOL;
      gR_T_1Min : BOOL;
      gF_T_1Min : BOOL;
      T_1SEC : REAL;
      del_T : REAL;
      NotHasRezervNU : BOOL;
      Reset_HasNU : BOOL;
      AI_A1_HA AT %QL0.8 : LREAL;
      AI_A1_HL AT %QL0.4 : LREAL;
      AI_A1_HW AT %QL0.10 : LREAL;
      AI_A1_LA AT %QL0.12 : LREAL;
      AI_A1_LL AT %QL0.5 : LREAL;
      AI_A1_LW AT %QL0.14 : LREAL;
      AI_A1_command AT %QW0.2 : UINT;
      AI_A1_newHA AT %QL0.9 : LREAL;
      AI_A1_newHL AT %QL0.6 : LREAL;
      AI_A1_newHW AT %QL0.11 : LREAL;
      AI_A1_newLA AT %QL0.13 : LREAL;
      AI_A1_newLL AT %QL0.7 : LREAL;
      AI_A1_newLW AT %QL0.15 : LREAL;
      AI_A1_status AT %QD0.1 : UDINT;
      AI_A1_value AT %QL0.3 : LREAL;
      AI_A2_HA AT %QL0.23 : LREAL;
      AI_A2_HL AT %QL0.19 : LREAL;
      AI_A2_HW AT %QL0.25 : LREAL;
      AI_A2_LA AT %QL0.27 : LREAL;
      AI_A2_LL AT %QL0.20 : LREAL;
      AI_A2_LW AT %QL0.29 : LREAL;
      AI_A2_command AT %QW0.17 : UINT;
      AI_A2_newHA AT %QL0.24 : LREAL;
      AI_A2_newHL AT %QL0.21 : LREAL;
      AI_A2_newHW AT %QL0.26 : LREAL;
      AI_A2_newLA AT %QL0.28 : LREAL;
      AI_A2_newLL AT %QL0.22 : LREAL;
      AI_A2_newLW AT %QL0.30 : LREAL;
      AI_A2_status AT %QD0.16 : UDINT;
      AI_A2_value AT %QL0.18 : LREAL;
      A1_10_err_mode AT %QW0.825 : UINT;
      A1_11_err_mode AT %QW0.826 : UINT;
      A1_12_err_mode AT %QW0.827 : UINT;
      A1_13_err_mode AT %QW0.828 : UINT;
      A1_14_err_mode AT %QW0.829 : UINT;
      A1_15_err_mode AT %QW0.830 : UINT;
      A1_1_err_mode AT %QW0.816 : UINT;
      A1_2_err_mode AT %QW0.817 : UINT;
      A1_3_err_mode AT %QW0.818 : UINT;
      A1_4_err_mode AT %QW0.819 : UINT;
      A1_5_err_mode AT %QW0.820 : UINT;
      A1_6_err_mode AT %QW0.821 : UINT;
      A1_7_err_mode AT %QW0.822 : UINT;
      A1_8_err_mode AT %QW0.823 : UINT;
      A1_9_err_mode AT %QW0.824 : UINT;
      A2_10_err_mode AT %QW0.840 : UINT;
      A2_11_err_mode AT %QW0.841 : UINT;
      A2_12_err_mode AT %QW0.842 : UINT;
      A2_13_err_mode AT %QW0.843 : UINT;
      A2_14_err_mode AT %QW0.844 : UINT;
      A2_15_err_mode AT %QW0.845 : UINT;
      A2_1_err_mode AT %QW0.831 : UINT;
      A2_2_err_mode AT %QW0.832 : UINT;
      A2_3_err_mode AT %QW0.833 : UINT;
      A2_4_err_mode AT %QW0.834 : UINT;
      A2_5_err_mode AT %QW0.835 : UINT;
      A2_6_err_mode AT %QW0.836 : UINT;
      A2_7_err_mode AT %QW0.837 : UINT;
      A2_8_err_mode AT %QW0.838 : UINT;
      A2_9_err_mode AT %QW0.839 : UINT;
      AI_0_dblValue AT %QL0.736 : LREAL;
      AI_10_dblValue AT %QL0.746 : LREAL;
      AI_11_dblValue AT %QL0.747 : LREAL;
      AI_12_dblValue AT %QL0.748 : LREAL;
      AI_13_dblValue AT %QL0.749 : LREAL;
      AI_14_dblValue AT %QL0.750 : LREAL;
      AI_15_dblValue AT %QL0.751 : LREAL;
      AI_16_dblValue AT %QL0.752 : LREAL;
      AI_17_dblValue AT %QL0.753 : LREAL;
      AI_18_dblValue AT %QL0.754 : LREAL;
      AI_19_dblValue AT %QL0.755 : LREAL;
      AI_1_dblValue AT %QL0.737 : LREAL;
      AI_20_dblValue AT %QL0.756 : LREAL;
      AI_21_dblValue AT %QL0.757 : LREAL;
      AI_22_dblValue AT %QL0.758 : LREAL;
      AI_23_dblValue AT %QL0.759 : LREAL;
      AI_24_dblValue AT %QL0.760 : LREAL;
      AI_25_dblValue AT %QL0.761 : LREAL;
      AI_26_dblValue AT %QL0.762 : LREAL;
      AI_27_dblValue AT %QL0.763 : LREAL;
      AI_28_dblValue AT %QL0.764 : LREAL;
      AI_29_dblValue AT %QL0.765 : LREAL;
      AI_2_dblValue AT %QL0.738 : LREAL;
      AI_30_dblValue AT %QL0.766 : LREAL;
      AI_31_dblValue AT %QL0.767 : LREAL;
      AI_32_dblValue AT %QL0.768 : LREAL;
      AI_33_dblValue AT %QL0.769 : LREAL;
      AI_34_dblValue AT %QL0.770 : LREAL;
      AI_35_dblValue AT %QL0.771 : LREAL;
      AI_36_dblValue AT %QL0.772 : LREAL;
      AI_37_dblValue AT %QL0.773 : LREAL;
      AI_38_dblValue AT %QL0.774 : LREAL;
      AI_39_dblValue AT %QL0.775 : LREAL;
      AI_3_dblValue AT %QL0.739 : LREAL;
      AI_40_dblValue AT %QL0.776 : LREAL;
      AI_41_dblValue AT %QL0.777 : LREAL;
      AI_42_dblValue AT %QL0.778 : LREAL;
      AI_43_dblValue AT %QL0.779 : LREAL;
      AI_44_dblValue AT %QL0.780 : LREAL;
      AI_45_dblValue AT %QL0.781 : LREAL;
      AI_46_dblValue AT %QL0.782 : LREAL;
      AI_47_dblValue AT %QL0.783 : LREAL;
      AI_48_dblValue AT %QL0.784 : LREAL;
      AI_49_dblValue AT %QL0.785 : LREAL;
      AI_4_dblValue AT %QL0.740 : LREAL;
      AI_50_dblValue AT %QL0.786 : LREAL;
      AI_51_dblValue AT %QL0.787 : LREAL;
      AI_52_dblValue AT %QL0.788 : LREAL;
      AI_53_dblValue AT %QL0.789 : LREAL;
      AI_54_dblValue AT %QL0.790 : LREAL;
      AI_55_dblValue AT %QL0.791 : LREAL;
      AI_56_dblValue AT %QL0.792 : LREAL;
      AI_57_dblValue AT %QL0.793 : LREAL;
      AI_58_dblValue AT %QL0.794 : LREAL;
      AI_59_dblValue AT %QL0.795 : LREAL;
      AI_5_dblValue AT %QL0.741 : LREAL;
      AI_60_dblValue AT %QL0.796 : LREAL;
      AI_61_dblValue AT %QL0.797 : LREAL;
      AI_62_dblValue AT %QL0.798 : LREAL;
      AI_63_dblValue AT %QL0.799 : LREAL;
      AI_64_dblValue AT %QL0.800 : LREAL;
      AI_65_dblValue AT %QL0.801 : LREAL;
      AI_66_dblValue AT %QL0.802 : LREAL;
      AI_67_dblValue AT %QL0.803 : LREAL;
      AI_68_dblValue AT %QL0.804 : LREAL;
      AI_69_dblValue AT %QL0.805 : LREAL;
      AI_6_dblValue AT %QL0.742 : LREAL;
      AI_70_dblValue AT %QL0.806 : LREAL;
      AI_71_dblValue AT %QL0.807 : LREAL;
      AI_72_dblValue AT %QL0.808 : LREAL;
      AI_73_dblValue AT %QL0.809 : LREAL;
      AI_74_dblValue AT %QL0.810 : LREAL;
      AI_75_dblValue AT %QL0.811 : LREAL;
      AI_76_dblValue AT %QL0.812 : LREAL;
      AI_77_dblValue AT %QL0.813 : LREAL;
      AI_78_dblValue AT %QL0.814 : LREAL;
      AI_79_dblValue AT %QL0.815 : LREAL;
      AI_7_dblValue AT %QL0.743 : LREAL;
      AI_8_dblValue AT %QL0.744 : LREAL;
      AI_9_dblValue AT %QL0.745 : LREAL;
      BS_Core1 AT %QD0.603 : REAL;
      BS_Core2 AT %QD0.675 : REAL;
      BS_Core3 AT %QD0.683 : REAL;
      BS_Core4 AT %QD0.709 : REAL;
      BS_FreeMemory AT %QD0.730 : REAL;
      BS_Temp1 AT %QD0.734 : REAL;
      BS_Temp2 AT %QD0.735 : REAL;
      DI_0_1_wValue AT %QD0.852 : UDINT;
      DI_10_11_wValue AT %QD0.857 : UDINT;
      DI_12_13_wValue AT %QD0.858 : UDINT;
      DI_14_15_wValue AT %QD0.859 : UDINT;
      DI_16_17_wValue AT %QD0.860 : UDINT;
      DI_18_19_wValue AT %QD0.861 : UDINT;
      DI_20_21_wValue AT %QD0.862 : UDINT;
      DI_2_3_wValue AT %QD0.853 : UDINT;
      DI_4_5_wValue AT %QD0.854 : UDINT;
      DI_6_7_wValue AT %QD0.855 : UDINT;
      DI_8_9_wValue AT %QD0.856 : UDINT;
      DO_0_wValue AT %QW0.846 : UINT;
      DO_1_wValue AT %QW0.847 : UINT;
      DO_2_wValue AT %QW0.848 : UINT;
      DO_3_wValue AT %QW0.849 : UINT;
      DO_4_wValue AT %QW0.850 : UINT;
      DO_5_wValue AT %QW0.851 : UINT;
      IM_Avom1_inCommand_ARM AT %QW0.43 : UINT;
      IM_Avom1_status AT %QD0.44 : UDINT;
      IM_Avom2_inCommand_ARM AT %QW0.45 : UINT;
      IM_Avom2_status AT %QD0.46 : UDINT;
      IM_Avom3_inCommand_ARM AT %QW0.47 : UINT;
      IM_Avom3_status AT %QD0.48 : UDINT;
      IM_Avom4_inCommand_ARM AT %QW0.49 : UINT;
      IM_Avom4_status AT %QD0.50 : UDINT;
      IM_Kran1_inCommand_ARM AT %QW0.31 : UINT;
      IM_Kran1_status AT %QD0.32 : UDINT;
      IM_Kran2_inCommand_ARM AT %QW0.35 : UINT;
      IM_Kran2_status AT %QD0.36 : UDINT;
      IM_Kran3_inCommand_ARM AT %QW0.37 : UINT;
      IM_Kran3_status AT %QD0.38 : UDINT;
      IM_Kran4_inCommand_ARM AT %QW0.33 : UINT;
      IM_Kran4_status AT %QD0.34 : UDINT;
      IM_Mv_inCommand_ARM AT %QW0.51 : UINT;
      IM_Mv_status AT %QD0.52 : UDINT;
      IM_Nu2_inCommand_ARM AT %QW0.41 : UINT;
      IM_Nu2_status AT %QD0.42 : UDINT;
      IM_Nu_inCommand_ARM AT %QW0.39 : UINT;
      IM_Nu_status AT %QD0.40 : UDINT;
      IM_SectionSwitch1_inCommand_ARM AT %QW0.53 : UINT;
      IM_SectionSwitch1_status AT %QD0.54 : UDINT;
      IM_SingleSignals_SI0_status AT %QD0.55 : UDINT;
      IM_SingleSignals_SI1_status AT %QD0.56 : UDINT;
      IM_SingleSignals_SI2_status AT %QD0.57 : UDINT;
      IM_SingleSignals_SI3_status AT %QD0.58 : UDINT;
      IM_SingleSignals_SI4_status AT %QD0.59 : UDINT;
      IM_SingleSignals_SI5_status AT %QD0.60 : UDINT;
      IM_SingleSignals_SI6_status AT %QD0.61 : UDINT;
      Protections_AiP1_inCommand_ARM AT %QW0.74 : UINT;
      Protections_AiP1_status AT %QD0.75 : UDINT;
      Protections_AiP2_inCommand_ARM AT %QW0.76 : UINT;
      Protections_AiP2_status AT %QD0.77 : UDINT;
      Protections_AiP3_inCommand_ARM AT %QW0.78 : UINT;
      Protections_AiP3_status AT %QD0.79 : UDINT;
      Protections_Ap1_inCommand_ARM AT %QW0.72 : UINT;
      Protections_Ap1_status AT %QD0.73 : UDINT;
      Protections_DiP1_inCommand_ARM AT %QW0.62 : UINT;
      Protections_DiP1_status AT %QD0.63 : UDINT;
      Protections_DiP2_inCommand_ARM AT %QW0.64 : UINT;
      Protections_DiP2_status AT %QD0.65 : UDINT;
      Protections_DiP3_inCommand_ARM AT %QW0.66 : UINT;
      Protections_DiP3_status AT %QD0.67 : UDINT;
      Protections_DiP4_inCommand_ARM AT %QW0.68 : UINT;
      Protections_DiP4_status AT %QD0.69 : UDINT;
      Protections_DiP5_inCommand_ARM AT %QW0.70 : UINT;
      Protections_DiP5_status AT %QD0.71 : UDINT;
    END_VAR
    TASK task0(INTERVAL := T#5ms,PRIORITY := 0);
    PROGRAM instance0 WITH task0 : program0;
  END_RESOURCE
END_CONFIGURATION
